// TwinCAT 3 PLC project WPPruefstand
// ProgramVersion: 3.1.4022.1
// CompilerDefines: VISU_USEPROPERTYINFO
// libraries:
//   VisuElem3DPath, 3.5.6.0 (System)
//   VisuElemMeter, 3.5.6.0 (System)
//   VisuElems, 3.5.6.10 (System)
//   VisuElemsDateTime, 3.5.6.0 (System)
//   VisuElemsSpecialControls, 3.5.6.0 (System)
//   VisuElemsWinControls, 3.5.6.0 (System)
//   VisuElemTextEditor, 3.5.6.0 (System)
//   visuinputs, 3.5.6.0 (system)
//   VisuNativeControl, 3.5.6.0 (System)
//   Tc2_Standard, * (Beckhoff Automation GmbH)
//   Tc2_System, * (Beckhoff Automation GmbH)
//   Tc2_Utilities, * (Beckhoff Automation GmbH)
//   Tc3_Module, * (Beckhoff Automation GmbH)
//   VisuDialogs, * (System)
// project tree:
//   DUTs/ E_PowMeas.TcDUT (not stored), E_Press.TcDUT (not stored), E_TempSensVR10.TcDUT (not stored), E_TempSensPT100.TcDUT (not stored), E_IndexPowMeas.TcDUT (not stored), E_SMStatus.TcDUT, E_TempSensVR11.TcDUT, E_Terminals.TcDUT (not stored), ST_InputVar.TcDUT (not stored), ST_InputVar_PowMeas.TcDUT (not stored), ST_OutputVar.TcDUT, ST_PumpTime.TcDUT
//   / GlobalTextList.TcGTLO (not stored), PlcTask.TcTTO, Visualization Manager.TcVMO (not stored)
//   GVLs/ DigOutputs.TcGVL, HeatingCurve.TcGVL, AnaOutputs.TcGVL (not stored), PID.TcGVL, PowMeas.TcGVL (not stored), Pressures.TcGVL (not stored), PumpTiming.TcGVL, StateMachine.TcGVL (not stored), SysCheck.TcGVL, SysCheckParams.TcGVL, TempConvDat.TcGVL, Temperatures.TcGVL, TempSetpoints.TcGVL, TerminalErrorRT.TcGVL, TimeProgs.TcGVL
//   POUs/ CheckDivDInt.TcPOU, CheckDivLInt.TcPOU (not stored), CheckDivLReal.TcPOU (not stored), CheckDivReal.TcPOU, MAIN.TcPOU (not stored), P_GetTime.TcPOU (not stored)
//   POUs/Control/ FB_AuxHeatCont.TcPOU (not stored), FB_CyclingControl.TcPOU, P_ControlMain.TcPOU (not stored)
//   POUs/Control/TemperatureControl/ FB_PIDSuppTemp.TcPOU, FB_SimpleTempCont.TcPOU, F_GetTempSP.TcPOU (not stored), I_TempController.TcIO (not stored), P_SHSuppTempPID.TcPOU
//   POUs/ErrorHandling/ F_WriteErrLog.TcPOU (not stored), P_EmShutdownAll.TcPOU (not stored), P_EmShutdownBPumpRun.TcPOU, P_EmShutdownHCPumpRun.TcPOU (not stored), P_EmShutdownPumpsRun.TcPOU (not stored), P_EmShutdownMain.TcPOU (not stored), P_ErrorHandlingMain.TcPOU (not stored), P_WriteErrLog.TcPOU (not stored)
//   POUs/Initialize/ FB_InitPumpTimes.TcPOU, FB_ReadHeatCurve.TcPOU, FB_ReadNightMode.TcPOU, FB_ReadPressTab.TcPOU, FB_ReadPT100Tab.TcPOU, FB_ReadTempResTabVR11.TcPOU, P_InitMain.TcPOU, FB_ReadTempResTabVR10.TcPOU, FB_InitTimes.TcPOU (not stored)
//   POUs/Read/ F_LinSens.TcPOU, F_NTCSens.TcPOU (not stored), F_PowMeasPhase.TcPOU (not stored), P_PowMeas.TcPOU, P_ReadMain.TcPOU, P_TestVals.TcPOU (not stored)
//   POUs/SystemCheck/ F_CheckAmbTemp.TcPOU (not stored), F_CheckBrinePressure.TcPOU (not stored), F_CheckCompCycPress.TcPOU, F_CheckCompOutTemp.TcPOU, F_CheckHeatCirPress.TcPOU, F_CheckHeatCirTemp.TcPOU (not stored), F_CheckPhaseSeq.TcPOU (not stored), F_CheckSens.TcPOU (not stored), F_CheckTerm.TcPOU (not stored), P_SysCheckMain.TcPOU
//   POUs/Write/ F_ConvLinAnaOutp.TcPOU (not stored), F_PumpConvPercVolt.TcPOU (not stored), FB_RampPump.TcPOU (not stored), P_WriteMain.TcPOU
//   VISUs/ Vis_ManCont.TcVIS (not stored), StandardVis.TcVIS (not stored)

CONFIGURATION WPPruefstand
    RESOURCE PLC ON TwinCAT3
        TASK PlcTask(INTERVAL := T#10ms, PRIORITY := 20);
        PROGRAM MAIN WITH PlcTask : MAIN;
    END_RESOURCE
END_CONFIGURATION

// ---- DUTs/E_SMStatus.TcDUT
{attribute 'strict'}
TYPE E_SMStatus :
(Initialize,
Read,
SystemCheck,
Automatic,
Write,
Error);
END_TYPE

// ---- DUTs/E_TempSensVR11.TcDUT
TYPE E_TempSensVR11 : //all VR11 temperature sensors
(
	T1,		//Temperature after compression
	T2,		//Temperature before compression
	T3,		//Source temperature before evaporator
	T4,		//Temperature before expansion valve
	T5,		//Temperature before internal heating circuit pump
	T6,		//Temperature after auxiliary heater
	T8		//Source temperature after brine pump
);
END_TYPE

// ---- DUTs/ST_OutputVar.TcDUT
TYPE ST_OutputVar :
STRUCT

(*
nVarOutput = (fVar-fParaC)/fParaM)
*)	

	nVarOutput AT %Q*	:INT;	//Output to terminal
	fVal				:REAL;	//Output value as REAL/FLOAT/SINGLE
	
	fParaMaxOutp		:REAL	:= 10;			//slope of linear conversion -> 10V, 32767 bit (INT16)
	nParaMaxInt			:INT	:= 32767;	
	fParaC				:REAL	:= 0;			//offset of linear conversion
	
	fParaMaxVal			:REAL;	//Maximum value of output (e.g. 10V, 20mA)
	fParaMinVal			:REAL;	//Minimum value of output (e.g. 0V, 4mA)
	
END_STRUCT
END_TYPE

// ---- DUTs/ST_PumpTime.TcDUT
TYPE ST_PumpTime :
STRUCT
	tPre	:	TIME;	//time the pump runs before compressor start
	tPost	:	TIME;	//time the pump runs after compressor stop
	bFirst	:	BOOL;	//flag if pump is the first one to start
	tDelay	:	Time;	//time the pump starts after the first pump
END_STRUCT
END_TYPE

// ---- GVLs/DigOutputs.TcGVL
{attribute 'qualified_only'}
VAR_GLOBAL
	//contactors
	bOutpComp	AT	%Q*	:	BOOL:=FALSE;	//Activate compressor - default: false
	bOutpAH		AT	%Q*	:	BOOL:=FALSE;	//Activate auxiliary heater - default: false
	
	//Switching valve
	bSHDHWSwitchValv	AT	%Q*	:	BOOL;	//Control signal for switching valve - Space Heating/DHW
	
END_VAR

// ---- GVLs/HeatingCurve.TcGVL
VAR_GLOBAL
	HeatCurve	:	ARRAY[0..40,0..1] OF REAL;
END_VAR

// ---- GVLs/PID.TcGVL
VAR_GLOBAL
	fKp			:	REAL	:= 1;		//proportional gain
	fTi			:	REAL	:= 10;		//integration time
	fTd			:	REAL	:= 0;		//derivative time
	tSamp		:	TIME	:= T#100MS;	//sampling time
	
	fErrSum		:	REAL	:= 0;	//sum of errors
	
	//limits of control signal - 0..10V signal
	fOutpUpLim	:	REAL	:=	10;
	fOutpLowLim	:	REAL	:=	0;
END_VAR

// ---- GVLs/PumpTiming.TcGVL
VAR_GLOBAL
	stBPTime			:	ST_PumpTime;
	stIntHeatCirTime	:	ST_PumpTime;
	nMaxPre				:	DWORD;
END_VAR

// ---- GVLs/SysCheck.TcGVL
VAR_GLOBAL
	bTermErrRT	:	BOOL	:=	FALSE;
	bSensErr	:	BOOL	:=	FALSE;
	bAmbTemp	:	BOOL	:=	FALSE;
	bBP			:	BOOL	:=	FALSE;
	bHCP		:	BOOL	:=	FALSE;
	bCompCyc	:	BOOL	:=	FALSE;
	bPhaseSeqCh	:	BOOL	:=	FALSE;
	bHeatTemp	:	BOOL	:=	FALSE;
	bCompOut	:	BOOL	:=	FALSE;
END_VAR

// ---- GVLs/SysCheckParams.TcGVL
VAR_GLOBAL
	(*
		All values except maximum compressor outlet temperature, maximum water supply temperature and 
		maximum water return temperature are set as recommended by the manufacturer. 
	*)	

	fMaxAmbTemp			:	REAL	:=	35;		//maximum ambient temperature
	fMinAmbTemp			:	REAL	:=	-20;	//minimum ambient temperature
	
	fBPMinOff			:	REAL	:=	0.2;	//minimum brine circuit pressure
	fBPMinOn			:	REAL	:=	0.4;	//brine circuit pressure for heat pump restart
	
	fHPMax				:	REAL	:=	30;		//maximum high pressure for compression cycle
	fLPMin				:	REAL	:=	0.7;	//minimum low pressure for compression cycle
	
	fTempCompOutMax		:	REAL	:=	120;	//maximum compressor outlet temperature
	
	fHCPMinOff			:	REAL	:=	0.5;	//minimum heating circuit pressure
	fHCPMinOn			:	REAL	:=	0.7;	//heating circuit pressure for heat pump restart
	
	fTempHeatSuppMax	:	REAL	:=	65;		//maximum water supply temperature
	fTempHeatRetMax		:	REAL	:=	60;		//maximum water return temperature
END_VAR

// ---- GVLs/TempConvDat.TcGVL
VAR_GLOBAL
	//stTempSensTables	:	ST_TempSensTables;
	VR10	:	ARRAY[1..40,1..2] OF REAL;
	VR11	:	ARRAY[1..40,1..2] OF REAL;
END_VAR

// ---- GVLs/Temperatures.TcGVL
{attribute 'qualified_only'}
VAR_GLOBAL
	eTempSensVR10	:	E_TempSensVR10;	//VR10 temperature sensors
	eTempSensVR11	:	E_TempSensVR11;	//VR11 temperature sensors
	eTempSensPT100	:	E_TempSensPT100;	//PT100 temperature sensors
	
	stTempSensVR10	:	ARRAY[0..3] OF ST_InputVar;	//Structures corresponding to temperature sensor enumeration
	stTempSensVR11	:	ARRAY[0..6] OF ST_InputVar;
	stTempSensPT100	:	ARRAY[0..3] OF ST_InputVar;

(*
	//Internal temperature sensors
	//Names of temperatures according to installation manual
	stT1	:	ST_InputVar;	//Temperature after compression
	stT2	:	ST_InputVar;	//Temperature before compression
	stT3	:	ST_InputVar;	//Source temperature before evaporator
	stT4	:	ST_InputVar;	//Temperature before expansion valve
	stT5	:	ST_InputVar;	//Temperature before internal heating circuit pump
	stT6	:	ST_InputVar;	//Temperature after auxiliary heater
	stT8	:	ST_InputVar;	//Source temperature after brine pump
	stSP	:	ST_InputVar;	//Temperature of DHW storage tank
	stVF1	:	ST_InputVar;	//Temperature at the top of the space heating buffer tank
	stVF2	:	ST_InputVar;	//Temperature after external mixing valve
	stRF1	:	ST_InputVar;	//Temperature at the bottom of the space heating buffer tank
	
	//Additional temperature sensors
	stTEXPVEV	:	ST_InputVar;	//Temperature between expansion valve and evaporator
	stTSHEV		:	ST_InputVar;	//Temperature after evaporator
	stTCond		:	ST_InputVar;	//Temperature after condenser
	stTAmp		:	ST_InputCar;	//Ambient temperature
*)

END_VAR

// ---- GVLs/TempSetpoints.TcGVL
VAR_GLOBAL
	fDHWUpSP			:	REAL	:=	65;	//hot water temperature upper setpoint for DHW
	fDHWLowSP			:	REAL	:=	55;	//hot water temperature lower setpoint for DHW
	fSpaceHeatSP		:	REAL;			//water supply temperature setpoint for space heating
	fRoomSetpoint		:	REAL	:=	20;	//room temperature setpoint temperature
	fRoomSetpointNight	:	REAL	:=	15;	//room temperature setpoint for night mode
END_VAR

// ---- GVLs/TerminalErrorRT.TcGVL
VAR_GLOBAL
	//check if the real-time communication with the terminals reports errors
	//checks State of Working Counter: 
	//0 - valid real-time communication
	//1 - invalid real-time communication
	bTermRt		AT %I*	:	ARRAY[0..8] OF BOOL;
END_VAR

// ---- GVLs/TimeProgs.TcGVL
VAR_GLOBAL
	todNightModeStart	:	TOD;
	todNightModeEnd		:	TOD;
END_VAR

// ---- POUs/CheckDivDInt.TcPOU
// Implicitly generated code : DO NOT EDIT
FUNCTION CheckDivDInt : DINT
VAR_INPUT
	divisor:DINT;
END_VAR

// Implicitly generated code : Only an Implementation suggestion
IF divisor = 0 THEN
	CheckDivDInt:=1;
	StateMachine.bFault		:=	TRUE;
	StateMachine.nFault		:=	2;
	StateMachine.sFaultMess	:=	'Critical program error: division by 0';
	StateMachine.eStatus	:=	Error;
	P_EmShutdownAll();	//Execute emergency shutdown
ELSE
	CheckDivDInt:=divisor;
END_IF;

END_FUNCTION

// ---- POUs/CheckDivReal.TcPOU
// Implicitly generated code : DO NOT EDIT
FUNCTION CheckDivReal : REAL
VAR_INPUT
	divisor:REAL;
END_VAR

// Implicitly generated code : Only an Implementation suggestion
IF divisor = 0 THEN
	CheckDivReal:=1;
	StateMachine.bFault		:=	TRUE;
	StateMachine.nFault		:=	2;
	StateMachine.sFaultMess	:=	'Critical program error: division by 0';
	StateMachine.eStatus	:=	Error;
	P_EmShutdownAll();	//Execute emergency shutdown
ELSE
	CheckDivReal:=divisor;
END_IF;

END_FUNCTION

// ---- POUs/Control/FB_CyclingControl.TcPOU
FUNCTION_BLOCK FB_CyclingControl
VAR_INPUT
	nMaxStarts	:	USINT	:=	3;		//maximum number of startups per hour
	nMinRunTime	:	DWORD	:=	300;	//minimum run time in seconds
	nMinOffTime	:	DWORD	:=	300;	//minimum off time in seconds
END_VAR
VAR_OUTPUT
	bStartupOK	:	BOOL;
	bShutdownOK	:	BOOL;
END_VAR
VAR
	//Startup counter
	TimHour		:	TON;	//timer for 1h
	
	//run time | off time
	nLastStart	:	DWORD;
	nLastStop	:	DWORD;
	
	//Current time
	nCurTime	:	DWORD;
	
END_VAR

//Timer parameters
TimHour.PT	:=	T#1h;
TimHour.IN	:=	TRUE;
TimHour();
IF TimHour.Q THEN			//one hour has passed
	TimHour.IN	:=	FALSE;	//reset timer
	TimHour();
	StateMachine.nNumStart	:=	0;		//reset counter
END_IF

//last start and stop time in seconds
nLastStart	:=	DT_TO_DWORD(StateMachine.dtLastStart);
nLastStop	:=	DT_TO_DWORD(StateMachine.dtLastStop);

//Current time
nCurTime	:=	DT_TO_DWORD(StateMachine.dtCurTime);	//current time in seconds

//set startup flag
IF (StateMachine.nNumStart >= nMaxStarts) OR (NOT ((nCurTime - nLastStop) >= (nMinOffTime - PumpTiming.nMaxPre))) THEN
	//disable startup, if max. starts per hour are reached or minimum off time is violated
	bSTartupOK	:=	FALSE;
ELSE
	bStartupOK	:=	TRUE;
END_IF

//set shutdown flag
IF NOT ((nCurTime - nLastStart) >= nMinRunTime) THEN
	bShutdownOK :=	FALSE;
ELSE
	bShutdownOK :=	TRUE;
END_IF

END_FUNCTION_BLOCK

// ---- POUs/Control/TemperatureControl/FB_PIDSuppTemp.TcPOU
FUNCTION_BLOCK FB_PIDSuppTemp
VAR_INPUT
	fSetPoint	:	REAL;
END_VAR
VAR_OUTPUT
	fOutp		:	REAL;
END_VAR
VAR
	Tim			:	TON;
	
	fErr		:	REAL;			//current difference between setpoint and actual value
	fErrOld		:	REAL	:= 0;	//error in last cycle
	
	eVF2		:	E_TempSensVR10	:=	VF2;
END_VAR

Tim(PT:=PID.tSamp,IN:=TRUE);

IF Tim.Q THEN
	//calculate current difference
	fErr	:=	fSetPoint - Temperatures.stTempSensVR10[eVF2].fVal;

	//Anti-windup
	IF (fOutp < PID.fOutpUpLim) AND (fOutp > PID.fOutpLowLim) THEN
		PID.fErrSum	:=	PID.fErrSum + (fErr * (TIME_TO_REAL(PID.tSamp)/1000));	//Integrate
	END_IF

	//calculate output signal
	fOutp	:=	PID.fKp * (fErr + (1/PID.fTi) * PID.fErrSum + PID.fTd * ((fErr - fErrOld)/(TIME_TO_REAL(PID.tSamp) / 1000)));

	IF fOutp > PID.fOutpUpLim THEN
		fOutp	:= PID.fOutpUpLim;
	ELSIF fOutp < PID.fOutpLowLim THEN
		fOutp	:=	PID.fOutpLowLim;
	END_IF

	//save error
	fErrOld	:=	fErr;
	
	//reset timer
	Tim(IN:=FALSE);
END_IF

END_FUNCTION_BLOCK

// ---- POUs/Control/TemperatureControl/FB_SimpleTempCont.TcPOU
FUNCTION_BLOCK FB_SimpleTempCont IMPLEMENTS I_TempController
VAR_INPUT
	//maximum times
	tMaxTimeDHW		:	TIME	:=	T#40M;
	tMaxTimeSH		:	TIME	:=	T#20M;
END_VAR
VAR_OUTPUT
END_VAR
VAR
	eSP				:	E_TempSensVR10	:=	SP;
	eRF1			:	E_TempSensVR10	:=	RF1;
	eVF1			:	E_TempSensVR10	:=	VF1;
	eAmb			:	E_TempSensPT100	:=	TAmb;
	
	//flags demand
	bDemDHW			:	BOOL	:=	FALSE;	//DHW demand
	bDemSH			:	BOOL	:=	FALSE;	//Space heating demand
	bEarlyRech		:	BOOL	:=	FALSE;	//early recharching of space heating buffer tank
	
	//timers for parallel demand
	TimDHW			:	TON;
	TimSH			:	TON;
	
	//Compressor control values
	CompOpCont		:	BOOL	:=	FALSE;
	ValveModeCont	:	BOOL;
	
	fSHTempSP		:	REAL;
END_VAR

//get temperature setpoint from heating curve
fSHTempSP	:=	F_GetTempSP(fAmbTemp:=Temperatures.stTempSensPT100[eAmb].fVal);

//identify DHW demand
IF (Temperatures.stTempSensVR10[eSP].fVal < TempSetpoints.fDHWLowSP) THEN
	bDemDHW		:=	TRUE;	//temperature lower than low setpoint -> demand
END_IF
IF (Temperatures.stTempSensVR10[eSP].fVal > TempSetpoints.fDHWUpSP) THEN
	IF ((Temperatures.stTempSensVR10[eVF1].fVal < (TempSetpoints.fSpaceHeatSP + 2))) AND bDemDHW THEN
		bEarlyRech	:=	TRUE;
	END_IF
	bDemDHW	:=	FALSE;	//temperature higher than upper setpoint -> cancel demand
END_IF

//identify space heating demand
IF (Temperatures.stTempSensVR10[eVF1].fVal < TempSetpoints.fSpaceHeatSP) THEN
	bDemSH		:=	TRUE;
END_IF
IF (Temperatures.stTempSensVR10[eRF1].fVal > (TempSetpoints.fSpaceHeatSP + 2)) THEN
	bDemSH		:=	FALSE;
END_IF
IF (Temperatures.stTempSensVR10[eRF1].fVal > (TempSetpoints.fSpaceHeatSP + 2)) THEN
	bEarlyRech	:=	FALSE;
END_IF

//Set modes

//Switching valve mode: 
//True: space heating mode
//False: DHW mode	
IF bDemDHW AND (NOT bDemSH) THEN			//only DHW demand
	ValveModeCont	:=	FALSE;
	CompOpCont		:=	TRUE;
ELSIF bDemSH AND (NOT bDemDHW) THEN			//only space heating demand
	ValveModeCont	:=	TRUE;
	CompOpCont		:=	TRUE;
ELSIF (NOT bDemSH) AND (NOT bDemDHW) THEN	//no demand
	IF bEarlyRech THEN	//early recharging
		ValveModeCont	:=	TRUE;
		CompOpCont		:=	TRUE;
	ELSE
		CompOpCont		:=	FALSE;
	END_IF
ELSIF bDemSH AND bDemDHW THEN				//parallel demand
	CompOpCont		:= TRUE;
	IF (NOT ValveModeCont) AND TimDHW.Q THEN	//max. time DHW mode reached
		ValveModeCont	:=	TRUE;	//switch to space heating
	ELSIF ValveModeCont AND TimSH.Q THEN		//max. time SH mode reached
		ValveModeCont	:=	FALSE;	//switch to DHW
	END_IF	
END_IF

//Timing
TimDHW.PT	:=	tMaxTimeDHW;
TImSH.PT	:=	tMaxTimeSH;
TimDHW();
TimSH();
IF StateMachine.bCompRun THEN	//only when the compressor is actually running
	IF ValveModeCont THEN
		TimSH.IN	:=	TRUE;
		TimDHW.IN	:=	FALSE;
	ELSE
		TimSH.IN	:=	FALSE;
		TimDHW.IN	:=	TRUE;
	END_IF
ELSE
	TimSH.IN		:=	FALSE;
	TimDHW.IN		:=	FALSE;
END_IF

PROPERTY CompOp : BOOL
GET
CompOp	:=	CompOpCont;
END_GET
SET
CompOpCont	:=	CompOp;
END_SET
END_PROPERTY

PROPERTY SpaceHeatTempSP : REAL
GET
SpaceHeatTempSP	:=	fSHTempSP;
END_GET
SET
fSHTempSP	:=	SpaceHeatTempSP;
END_SET
END_PROPERTY

PROPERTY ValveMode : BOOL
GET
ValveMode	:=	ValveModeCont;
END_GET
SET
ValveModeCont	:= ValveMode;
END_SET
END_PROPERTY

END_FUNCTION_BLOCK

// ---- POUs/Control/TemperatureControl/P_SHSuppTempPID.TcPOU
PROGRAM P_SHSuppTempPID
VAR
	eTAmb			:	E_TempSensPT100	:=	TAmb;	//ambient temperature
	fTAmbMax		:	REAL			:=	21;		//maximum ambient temperature before space heating is switched off
	fbPIDSuppTemp	:	FB_PIDSuppTemp;				//PID controller
	fPIDOutp		:	REAL;						//control signal from PID
	bAct			:	BOOL			:=	True;	//space heating active
END_VAR

IF Temperatures.stTempSensPT100[eTAmb].fVal > (fTAmbMax + 1) THEN
	bAct	:=	FALSE;
ELSIF Temperatures.stTempSensPT100[eTAmb].fVal < (fTAmbMax - 1) THEN
	bAct	:=	TRUE;
END_IF
	
IF bAct THEN
	//run external heating circuit pump
	StateMachine.bExtHeatCPump	:=	TRUE;

	//execute PID Control
	fbPIDSuppTemp(fSetPoint:=TempSetpoints.fSpaceHeatSP);
	fPIDOutp	:=	fbPIDSuppTemp.fOutp;

	//pass control signal to mixing valve
	StateMachine.fMixVal	:=	fPIDOutp;
ELSE
	StateMachine.bExtHeatCPump	:=	FALSE;
END_IF

END_PROGRAM

// ---- POUs/ErrorHandling/P_EmShutdownBPumpRun.TcPOU
PROGRAM P_EmShutdownBPumpRun
VAR
END_VAR

//shut down all components except brine pump

StateMachine.bCompRun		:=	FALSE;
DigOutputs.bOutpComp		:=	FALSE;

StateMachine.bAuxHeatOp		:=	FALSE;
DigOutputs.bOutpAH			:=	FALSE;

StateMachine.bBrinePump		:=	TRUE;
AnaOutputs.stOutpBP.fVal	:=	10;
AnaOutputs.stOutpBP			:=	F_ConvLinAnaOutp(stOutput:=AnaOutputs.stOutpBP);

StateMachine.bIntHeatCPump	:=	FALSE;
AnaOutputs.stOutpIntHP.fVal	:=	0.75;	//0.75 Volt: Pump stop
AnaOutputs.stOutpIntHP		:=	F_ConvLinAnaOutp(stOutput:=AnaOutputs.stOutpIntHP);

StateMachine.bExtHeatCPump	:=	TRUE;
AnaOutputs.stOutpExtHP.fVal	:=	10;	
AnaOutputs.stOutpExtHP			:=	F_ConvLinAnaOutp(stOutput:=AnaOutputs.stOutpExtHP);

StateMachine.bCircPump		:=	TRUE;

END_PROGRAM

// ---- POUs/Initialize/FB_InitPumpTimes.TcPOU
FUNCTION_BLOCK FB_InitPumpTimes
VAR_INPUT
	tBP_Pre				:	TIME	:=	T#1M;
	tIntHeatCir_Pre		:	TIME	:=	T#1M;
	tBP_Post			:	TIME	:=	T#5M;
	tIntHeatCir_Post	:	TIME	:=	T#30M;
END_VAR
VAR_OUTPUT
	bReady	:	BOOL	:=	False;
END_VAR
VAR
END_VAR

//write to GVL
PumpTiming.stBPTime.tPre			:=	tBP_Pre;
PumpTiming.stIntHeatCirTime.tPre	:=	tIntHeatCir_Pre;
PumpTiming.stBPTime.tPost			:=	tBP_Post;
PumpTiming.stIntHeatCirTime.tPost	:=	tIntHeatCir_Post;

//find first one to start and calculate delays
IF (tBP_Pre > tIntHeatCir_Pre) THEN
	PumpTiming.stBPTime.bFirst			:=	TRUE;
	PumpTiming.stBPTime.tDelay			:=	T#0MS;
	PumpTiming.stIntHeatCirTime.tDelay	:=	tBP_Pre - tIntHeatCir_Pre;
	PumpTiming.nMaxPre					:=	(TIME_TO_DWORD(tBP_Pre)/1000);
ELSE
	PumpTiming.stIntHeatCirTime.bFirst	:=	TRUE;
	PumpTiming.stIntHeatCirTime.tDelay	:=	T#0MS;
	PumpTiming.stBPTime.tDelay			:=	tIntHeatCir_Pre - tBP_Pre;
	PumpTiming.nMaxPre					:=	(TIME_TO_DWORD(tIntHeatCir_Pre)/1000);
END_IF

bReady	:=	TRUE;

END_FUNCTION_BLOCK

// ---- POUs/Initialize/FB_ReadHeatCurve.TcPOU
FUNCTION_BLOCK FB_ReadHeatCurve
VAR_INPUT
	bExecute		:	BOOL	:= FALSE;
END_VAR
VAR_OUTPUT
	bCompleted		:	BOOL	:=	FALSE;
	bError			:	BOOL	:=	FALSE;
END_VAR
VAR
	fbFileOpen		:	FB_FileOpen;
	fbFileGets		:	FB_FileGets;
	fbReader		:	FB_CSVMemBufferReader;
	fbFileClose		:	FB_FileClose;
	sCSVPath		:	STRING	:=	'D:\cve-mme\WpPruefstandData\Heizkurve.csv';	//Path to csv file
	hFile			:	UINT;
	bEOF			:	BOOL	:=	FALSE;
	Step			:	DWORD	:=	0;
	sLine			:	STRING;	//Line read by fbFileGets
	nLine			:	UINT	:=	0;
END_VAR

CASE Step OF
	
0:	//Standby mode
	IF bExecute THEN
		bExecute	:=	FALSE; //reset to defaults
		hFile		:=	0;
		bEOF		:=	FALSE;
		bCompleted	:=	FALSE;
		bError		:=	FALSE;
		sLine		:=	'';
		nLine		:=	0;
		Step		:=	1; //start program
	END_IF

1:	//Open file
	fbFileOpen(sNetId:='', sPathName:=sCSVPath, nMode:=FOPEN_MODEREAD OR FOPEN_MODETEXT,
		ePath:=PATH_GENERIC, tTimeout:=T#5s, bExecute:=TRUE);
	Step	:=	Step + 1;

2:
	fbFileOpen(bExecute:=FALSE);
	IF NOT fbFileOpen.bBusy THEN
		IF NOT fbFileOpen.bError THEN
			//Store file handle
			hFile	:=	fbFileOpen.hFile;
			Step	:=	Step + 1;
		ELSE
			Step	:=	90;	
		END_IF
	END_IF

3:	//Read csv file
	fbFileGets(sNetId:='', hFile:=hFile, bExecute:=TRUE, tTimeout:=T#5S);
	nLine	:=	nLine + 1;
	Step	:=	Step + 1;

4:
	fbFileGets(bExecute:=FALSE);
	IF NOT fbFileGets.bBusy THEN
		IF NOT (nLine = 1) THEN //Header -> jump to next line
			IF NOT fbFileGets.bError THEN
				IF fbFileGets.bEOF THEN
					Step	:=	10; //Reached end of file
				ELSE
					sLine	:=	fbFileGets.sLine; //store line
					IF RIGHT(sLine,1) = '$L' THEN
						sLine	:=	REPLACE(sLINE, '$R$L', 2, LEN(sLine)); //restore CRLF characters
					END_IF
					Step	:=	Step + 1;
				END_IF
			ELSE
				Step	:=	90;
			END_IF
		ELSE
			Step	:=	3;
		END_IF
	END_IF
	
5:	//Parse line
	
	fbReader.eCmd	:=	eEnumCmd_First;	//Read first value (ambient temperature)
	fbReader(pBuffer:=ADR(sLine), cbBuffer:=SIZEOF(sLine));
	
	IF fbReader.bOk THEN
		HeatingCurve.HeatCurve[nLine-2,0] := STRING_TO_REAL(fbReader.getValue);	//account for header
	ELSE
		Step	:=	90;
	END_IF	
	
	fbReader.eCmd	:=	eEnumCmd_Next;	//Read next value (temperature setpoint)
	fbReader(pBuffer:=ADR(sLine), cbBuffer:=SIZEOF(sLine));
	
	IF fbReader.bOk THEN
		HeatingCurve.HeatCurve[nLine-2,1] := STRING_TO_REAL(fbReader.getValue); //account for header
	ELSE
		Step	:=	90;
	END_IF
	
	//Read next line
	Step	:=	3;
	
10:	//end of csv file
	IF (hFile <> 0) THEN
		Step	:=	20; //close file
	END_IF
	
20:	//close csv file
	fbFileClose(bExecute:=FALSE);
	fbFileClose(sNetId:='', hFile:=hFile, bExecute:=TRUE, tTimeout:=T#5S);
	Step	:=	21;
	
21:	
	fbFileClose(bExecute:=FALSE);
	IF NOT fbFileClose.bBusy THEN
		step	:=	0;	//Standby mode
		bCompleted	:=	TRUE;
	END_IF
	
90:	//TODO: Error handling
	bError	:=	TRUE;
	IF (hFile <> 0) THEN
		Step	:=	20;	//close file
	END_IF

END_CASE

END_FUNCTION_BLOCK

// ---- POUs/Initialize/FB_ReadNightMode.TcPOU
FUNCTION_BLOCK FB_ReadNightMode
VAR_INPUT
	bExecute		:	BOOL	:= FALSE;
END_VAR
VAR_OUTPUT
	bCompleted		:	BOOL	:=	FALSE;
	bError			:	BOOL	:=	FALSE;
END_VAR
VAR
	fbFileOpen		:	FB_FileOpen;
	fbFileGets		:	FB_FileGets;
	fbReader		:	FB_CSVMemBufferReader;
	fbFileClose		:	FB_FileClose;
	sCSVPath		:	STRING	:=	'D:\cve-mme\WpPruefstandData\NightMode.csv';	//Path to csv file
	hFile			:	UINT;
	bEOF			:	BOOL	:=	FALSE;
	Step			:	DWORD	:=	0;
	sLine			:	STRING;	//Line read by fbFileGets
	nLine			:	UINT	:=	0;
	nHourStart		:	USINT;
	nHourStop		:	USINT;
	nMinStart		:	USINT;
	nMinStop		:	USINT;
	nStartTime		:	UDINT;	//Start time in ms
	nStopTime		:	UDINT;	//Stop time in ms
END_VAR

CASE Step OF
	
0:	//Standby mode
	IF bExecute THEN
		bExecute	:=	FALSE; //reset to defaults
		hFile		:=	0;
		bEOF		:=	FALSE;
		bCompleted	:=	FALSE;
		bError		:=	FALSE;
		sLine		:=	'';
		nLine		:=	0;
		Step		:=	1; //start program
	END_IF

1:	//Open file
	fbFileOpen(sNetId:='', sPathName:=sCSVPath, nMode:=FOPEN_MODEREAD OR FOPEN_MODETEXT,
		ePath:=PATH_GENERIC, tTimeout:=T#5s, bExecute:=TRUE);
	Step	:=	Step + 1;

2:
	fbFileOpen(bExecute:=FALSE);
	IF NOT fbFileOpen.bBusy THEN
		IF NOT fbFileOpen.bError THEN
			//Store file handle
			hFile	:=	fbFileOpen.hFile;
			Step	:=	Step + 1;
		ELSE
			Step	:=	90;	
		END_IF
	END_IF

3:	//Read csv file
	fbFileGets(sNetId:='', hFile:=hFile, bExecute:=TRUE, tTimeout:=T#5S);
	nLine	:=	nLine + 1;
	Step	:=	Step + 1;

4:
	fbFileGets(bExecute:=FALSE);
	IF NOT fbFileGets.bBusy THEN
		IF NOT (nLine = 1) THEN //Header -> jump to next line
			IF NOT fbFileGets.bError THEN
				IF fbFileGets.bEOF THEN
					Step	:=	10; //Reached end of file
				ELSE
					sLine	:=	fbFileGets.sLine; //store line
					IF RIGHT(sLine,1) = '$L' THEN
						sLine	:=	REPLACE(sLINE, '$R$L', 2, LEN(sLine)); //restore CRLF characters
					END_IF
					Step	:=	Step + 1;
				END_IF
			ELSE
				Step	:=	90;
			END_IF
		ELSE
			Step	:=	3;
		END_IF
	END_IF
	
5:	//Parse line
	fbReader.eCmd	:=	eEnumCmd_First;	//Read first value (identifier)
	fbReader(pBuffer:=ADR(sLine), cbBuffer:=SIZEOF(sLine));
	
	fbReader.eCmd	:=	eEnumCmd_Next;	//Read next value (hour)
	fbReader(pBuffer:=ADR(sLine), cbBuffer:=SIZEOF(sLine));
	
	IF fbReader.bOk THEN
		IF (nLine = 2) THEN
			nHourStart	:=	STRING_TO_USINT(fbReader.getValue);
		ELSIF (nLine = 3) THEN
			nHourStop	:=	STRING_TO_USINT(fbReader.getValue);
		ELSE
			Step	:=	90;
		END_IF
	ELSE
		Step	:=	90;
	END_IF	
	
	fbReader.eCmd	:=	eEnumCmd_Next;	//Read next value (minute)
	fbReader(pBuffer:=ADR(sLine), cbBuffer:=SIZEOF(sLine));
	
	IF fbReader.bOk THEN
		IF (nLine = 2) THEN
			nMinStart	:=	STRING_TO_USINT(fbReader.getValue);
		ELSIF (nLine = 3) THEN
			nMinStop	:=	STRING_TO_USINT(fbReader.getValue);
		ELSE
			Step	:=	90;
		END_IF
	ELSE
		Step	:=	90;
	END_IF
	
	//Read next line
	Step	:=	3;
	
10:	//end of csv file
	IF (hFile <> 0) THEN
		Step	:=	20; //close file
	END_IF
	
20:	//close csv file
	fbFileClose(bExecute:=FALSE);
	fbFileClose(sNetId:='', hFile:=hFile, bExecute:=TRUE, tTimeout:=T#5S);
	Step	:=	21;
	
21:	
	fbFileClose(bExecute:=FALSE);
	IF NOT fbFileClose.bBusy THEN
		//convert data and write to GVL
		nStartTime	:=	nHourStart * 3600 * 1000 + nMinStart * 60 * 1000;
		nStopTime	:=	nHourStop * 3600 * 1000 + nMinStop * 60 * 1000;
		TimeProgs.todNightModeStart	:=	UDINT_TO_TOD(nStartTime);
		TimeProgs.todNightModeEnd	:=	UDINT_TO_TOD(nStopTime);
	
		step	:=	0;	//Standby mode
		bCompleted	:=	TRUE;
	END_IF
	
90:	//TODO: Error handling
	bError	:=	TRUE;
	IF (hFile <> 0) THEN
		Step	:=	20;	//close file
	END_IF

END_CASE

END_FUNCTION_BLOCK

// ---- POUs/Initialize/FB_ReadPressTab.TcPOU
FUNCTION_BLOCK FB_ReadPressTab
VAR_INPUT
	bExecute		:	BOOL	:= FALSE;
END_VAR
VAR_OUTPUT
	bCompleted		:	BOOL	:=	FALSE;
	bError			:	BOOL	:=	FALSE;
END_VAR
VAR
	fbFileOpen		:	FB_FileOpen;
	fbFileGets		:	FB_FileGets;
	fbReader		:	FB_CSVMemBufferReader;
	fbFileClose		:	FB_FileClose;
	sCSVPath		:	STRING	:=	'D:\cve-mme\WpPruefstandData\PressureDat.csv';	//Path to csv file
	hFile			:	UINT;
	bEOF			:	BOOL	:=	FALSE;
	Step			:	DWORD	:=	0;
	sLine			:	STRING;	//Line read by fbFileGets
	nLine			:	UINT	:=	0;
	nIndSens		:	INT;
	stSensName		:	String;
END_VAR

CASE Step OF
	
0:	//Standby mode
	IF bExecute THEN
		bExecute	:=	FALSE; //reset to defaults
		hFile		:=	0;
		bEOF		:=	FALSE;
		bCompleted	:=	FALSE;
		bError		:=	FALSE;
		sLine		:=	'';
		nLine		:=	0;
		Step		:=	1; //start program
	END_IF

1:	//Open file
	fbFileOpen(sNetId:='', sPathName:=sCSVPath, nMode:=FOPEN_MODEREAD OR FOPEN_MODETEXT,
		ePath:=PATH_GENERIC, tTimeout:=T#5s, bExecute:=TRUE);
	Step	:=	Step + 1;

2:
	fbFileOpen(bExecute:=FALSE);
	IF NOT fbFileOpen.bBusy THEN
		IF NOT fbFileOpen.bError THEN
			//Store file handle
			hFile	:=	fbFileOpen.hFile;
			Step	:=	Step + 1;
		ELSE
			Step	:=	90;	
		END_IF
	END_IF

3:	//Read csv file
	fbFileGets(sNetId:='', hFile:=hFile, bExecute:=TRUE, tTimeout:=T#5S);
	nLine	:=	nLine + 1;
	Step	:=	Step + 1;

4:
	fbFileGets(bExecute:=FALSE);
	IF NOT fbFileGets.bBusy THEN
		IF NOT (nLine = 1) THEN //Header -> jump to next line
			IF NOT fbFileGets.bError THEN
				IF fbFileGets.bEOF THEN
					Step	:=	10; //Reached end of file
				ELSE
					sLine	:=	fbFileGets.sLine; //store line
					IF RIGHT(sLine,1) = '$L' THEN
						sLine	:=	REPLACE(sLINE, '$R$L', 2, LEN(sLine)); //restore CRLF characters
					END_IF
					Step	:=	Step + 1;
				END_IF
			ELSE
				Step	:=	90;
			END_IF
		ELSE
			Step	:=	3;
		END_IF
	END_IF
	
5:	//Parse line
	fbReader.eCmd	:=	eEnumCmd_First;	//Read first value (identifier)
	fbReader(pBuffer:=ADR(sLine), cbBuffer:=SIZEOF(sLine));
	
	IF fbReader.bOk THEN
		stSensName	:= fbReader.getValue;	//identify index of current sensor
		IF (FIND(str1:=stSensName, str2:='HP') <> 0) THEN
			Pressures.ePress	:=	HP;
		ELSIF (FIND(str1:=stSensName, str2:='LP') <> 0) THEN
			Pressures.ePress	:=	LP;
		ELSIF (FIND(str1:=stSensName, str2:='HCP') <> 0) THEN
			Pressures.ePress	:=	HCP;
		ELSIF (FIND(str1:=stSensName, str2:='BP') <> 0) THEN
			Pressures.ePress	:=	BP;
		END_IF
		nIndSens	:=	Pressures.ePress;
	ELSE
		Step	:=	90;
	END_IF	
	
	fbReader.eCmd	:=	eEnumCmd_Next;	//Read next value (slope)
	fbReader(pBuffer:=ADR(sLine), cbBuffer:=SIZEOF(sLine));
	
	IF fbReader.bOk THEN
		Pressures.stPress[nIndSens].fParaM := STRING_TO_REAL(fbReader.getValue);
	ELSE
		Step	:=	90;
	END_IF	
	
	fbReader.eCmd	:=	eEnumCmd_Next;	//Read next value (offset)
	fbReader(pBuffer:=ADR(sLine), cbBuffer:=SIZEOF(sLine));
	
	IF fbReader.bOk THEN
		Pressures.stPress[nIndSens].fParaC := STRING_TO_REAL(fbReader.getValue); //account for header
	ELSE
		Step	:=	90;
	END_IF
	
	fbReader.eCmd	:=	eEnumCmd_Next;	//Read next value (maximum value)
	fbReader(pBuffer:=ADR(sLine), cbBuffer:=SIZEOF(sLine));
	
	IF fbReader.bOk THEN
		Pressures.stPress[nIndSens].fParaMaxVal := STRING_TO_REAL(fbReader.getValue); //account for header
	ELSE
		Step	:=	90;
	END_IF
	
	fbReader.eCmd	:=	eEnumCmd_Next;	//Read next value (minimum value)
	fbReader(pBuffer:=ADR(sLine), cbBuffer:=SIZEOF(sLine));
	
	IF fbReader.bOk THEN
		Pressures.stPress[nIndSens].fParaMinVal := STRING_TO_REAL(fbReader.getValue); //account for header
	ELSE
		Step	:=	90;
	END_IF
	
	//Read next line
	Step	:=	3;
	
10:	//end of csv file
	IF (hFile <> 0) THEN
		Step	:=	20; //close file
	END_IF
	
20:	//close csv file
	fbFileClose(bExecute:=FALSE);
	fbFileClose(sNetId:='', hFile:=hFile, bExecute:=TRUE, tTimeout:=T#5S);
	Step	:=	21;
	
21:	
	fbFileClose(bExecute:=FALSE);
	IF NOT fbFileClose.bBusy THEN
		step	:=	0;	//Standby mode
		bCompleted	:=	TRUE;
	END_IF
	
90:	//TODO: Error handling
	bError	:=	TRUE;
	IF (hFile <> 0) THEN
		Step	:=	20;	//close file
	END_IF

END_CASE

END_FUNCTION_BLOCK

// ---- POUs/Initialize/FB_ReadPT100Tab.TcPOU
FUNCTION_BLOCK FB_ReadPT100Tab
VAR_INPUT
	bExecute		:	BOOL	:= FALSE;
END_VAR
VAR_OUTPUT
	bCompleted		:	BOOL	:=	FALSE;
	bError			:	BOOL	:=	FALSE;
END_VAR
VAR
	fbFileOpen		:	FB_FileOpen;
	fbFileGets		:	FB_FileGets;
	fbReader		:	FB_CSVMemBufferReader;
	fbFileClose		:	FB_FileClose;
	sCSVPath		:	STRING	:=	'D:\cve-mme\WpPruefstandData\PT100Dat.csv';	//Path to csv file
	hFile			:	UINT;
	bEOF			:	BOOL	:=	FALSE;
	Step			:	DWORD	:=	0;
	sLine			:	STRING;	//Line read by fbFileGets
	nLine			:	UINT	:=	0;
	nIndSens		:	INT;
	stSensName		:	String;
END_VAR

CASE Step OF
	
0:	//Standby mode
	IF bExecute THEN
		bExecute	:=	FALSE; //reset to defaults
		hFile		:=	0;
		bEOF		:=	FALSE;
		bCompleted	:=	FALSE;
		bError		:=	FALSE;
		sLine		:=	'';
		nLine		:=	0;
		Step		:=	1; //start program
	END_IF

1:	//Open file
	fbFileOpen(sNetId:='', sPathName:=sCSVPath, nMode:=FOPEN_MODEREAD OR FOPEN_MODETEXT,
		ePath:=PATH_GENERIC, tTimeout:=T#5s, bExecute:=TRUE);
	Step	:=	Step + 1;

2:
	fbFileOpen(bExecute:=FALSE);
	IF NOT fbFileOpen.bBusy THEN
		IF NOT fbFileOpen.bError THEN
			//Store file handle
			hFile	:=	fbFileOpen.hFile;
			Step	:=	Step + 1;
		ELSE
			Step	:=	90;	
		END_IF
	END_IF

3:	//Read csv file
	fbFileGets(sNetId:='', hFile:=hFile, bExecute:=TRUE, tTimeout:=T#5S);
	nLine	:=	nLine + 1;
	Step	:=	Step + 1;

4:
	fbFileGets(bExecute:=FALSE);
	IF NOT fbFileGets.bBusy THEN
		IF NOT (nLine = 1) THEN //Header -> jump to next line
			IF NOT fbFileGets.bError THEN
				IF fbFileGets.bEOF THEN
					Step	:=	10; //Reached end of file
				ELSE
					sLine	:=	fbFileGets.sLine; //store line
					IF RIGHT(sLine,1) = '$L' THEN
						sLine	:=	REPLACE(sLINE, '$R$L', 2, LEN(sLine)); //restore CRLF characters
					END_IF
					Step	:=	Step + 1;
				END_IF
			ELSE
				Step	:=	90;
			END_IF
		ELSE
			Step	:=	3;
		END_IF
	END_IF
	
5:	//Parse line
	fbReader.eCmd	:=	eEnumCmd_First;	//Read first value (identifier)
	fbReader(pBuffer:=ADR(sLine), cbBuffer:=SIZEOF(sLine));
	
	IF fbReader.bOk THEN
		stSensName	:= fbReader.getValue;	//identify index of current sensor
		IF (FIND(str1:=stSensName, str2:='TExpVEv') <> 0) THEN
			Temperatures.eTempSensPT100	:=	TExpVEv;
		ELSIF (FIND(str1:=stSensName, str2:='TShEv') <> 0) THEN
			Temperatures.eTempSensPT100	:=	TShEv;
		ELSIF (FIND(str1:=stSensName, str2:='TCond') <> 0) THEN
			Temperatures.eTempSensPT100	:=	TCond;
		ELSIF (FIND(str1:=stSensName, str2:='TAmb') <> 0) THEN
			Temperatures.eTempSensPT100	:=	TAmb;
		END_IF
		nIndSens	:=	Temperatures.eTempSensPT100;
	ELSE
		Step	:=	90;
	END_IF	
	
	fbReader.eCmd	:=	eEnumCmd_Next;	//Read next value (slope)
	fbReader(pBuffer:=ADR(sLine), cbBuffer:=SIZEOF(sLine));
	
	IF fbReader.bOk THEN
		Temperatures.stTempSensPT100[nIndSens].fParaM := STRING_TO_REAL(fbReader.getValue);
	ELSE
		Step	:=	90;
	END_IF	
	
	fbReader.eCmd	:=	eEnumCmd_Next;	//Read next value (offset)
	fbReader(pBuffer:=ADR(sLine), cbBuffer:=SIZEOF(sLine));
	
	IF fbReader.bOk THEN
		Temperatures.stTempSensPT100[nIndSens].fParaC := STRING_TO_REAL(fbReader.getValue); //account for header
	ELSE
		Step	:=	90;
	END_IF
	
	fbReader.eCmd	:=	eEnumCmd_Next;	//Read next value (maximum value)
	fbReader(pBuffer:=ADR(sLine), cbBuffer:=SIZEOF(sLine));
	
	IF fbReader.bOk THEN
		Temperatures.stTempSensPT100[nIndSens].fParaMaxVal := STRING_TO_REAL(fbReader.getValue); //account for header
	ELSE
		Step	:=	90;
	END_IF
	
	fbReader.eCmd	:=	eEnumCmd_Next;	//Read next value (minimum value)
	fbReader(pBuffer:=ADR(sLine), cbBuffer:=SIZEOF(sLine));
	
	IF fbReader.bOk THEN
		Temperatures.stTempSensPT100[nIndSens].fParaMinVal := STRING_TO_REAL(fbReader.getValue);
	ELSE
		Step	:=	90;
	END_IF
	
	//Read next line
	Step	:=	3;
	
10:	//end of csv file
	IF (hFile <> 0) THEN
		Step	:=	20; //close file
	END_IF
	
20:	//close csv file
	fbFileClose(bExecute:=FALSE);
	fbFileClose(sNetId:='', hFile:=hFile, bExecute:=TRUE, tTimeout:=T#5S);
	Step	:=	21;
	
21:	
	fbFileClose(bExecute:=FALSE);
	IF NOT fbFileClose.bBusy THEN
		step	:=	0;	//Standby mode
		bCompleted	:=	TRUE;
	END_IF
	
90:	//TODO: Error handling
	bError	:=	TRUE;
	IF (hFile <> 0) THEN
		Step	:=	20;	//close file
	END_IF

END_CASE

END_FUNCTION_BLOCK

// ---- POUs/Initialize/FB_ReadTempResTabVR11.TcPOU
FUNCTION_BLOCK FB_ReadTempResTabVR11
VAR_INPUT
	bExecute		:	BOOL	:= FALSE;
END_VAR
VAR_OUTPUT
	bCompleted		:	BOOL	:=	FALSE;
	bError			:	BOOL	:=	FALSE;
END_VAR
VAR
	fbFileOpen		:	FB_FileOpen;
	fbFileGets		:	FB_FileGets;
	fbReader		:	FB_CSVMemBufferReader;
	fbFileClose		:	FB_FileClose;
	sCSVPath		:	STRING	:=	'D:\cve-mme\WpPruefstandData\KennlinieVR11.csv';	//Path to csv file
	hFile			:	UINT;
	bEOF			:	BOOL	:=	FALSE;
	Step			:	DWORD	:=	0;
	sLine			:	STRING;	//Line read by fbFileGets
	nLine			:	UINT	:=	0;
END_VAR

CASE Step OF
	
0:	//Standby mode
	IF bExecute THEN
		bExecute	:=	FALSE; //reset to defaults
		hFile		:=	0;
		bEOF		:=	FALSE;
		bCompleted	:=	FALSE;
		bError		:=	FALSE;
		sLine		:=	'';
		nLine		:=	0;
		Step		:=	1; //start program
	END_IF

1:	//Open file
	fbFileOpen(sNetId:='', sPathName:=sCSVPath, nMode:=FOPEN_MODEREAD OR FOPEN_MODETEXT,
		ePath:=PATH_GENERIC, tTimeout:=T#5s, bExecute:=TRUE);
	Step	:=	Step + 1;

2:
	fbFileOpen(bExecute:=FALSE);
	IF NOT fbFileOpen.bBusy THEN
		IF NOT fbFileOpen.bError THEN
			//Store file handle
			hFile	:=	fbFileOpen.hFile;
			Step	:=	Step + 1;
		ELSE
			Step	:=	90;	
		END_IF
	END_IF

3:	//Read csv file
	fbFileGets(sNetId:='', hFile:=hFile, bExecute:=TRUE, tTimeout:=T#5S);
	nLine	:=	nLine + 1;
	Step	:=	Step + 1;

4:
	fbFileGets(bExecute:=FALSE);
	IF NOT fbFileGets.bBusy THEN
		IF NOT (nLine = 1) THEN //Header -> jump to next line
			IF NOT fbFileGets.bError THEN
				IF fbFileGets.bEOF THEN
					Step	:=	10; //Reached end of file
				ELSE
					sLine	:=	fbFileGets.sLine; //store line
					IF RIGHT(sLine,1) = '$L' THEN
						sLine	:=	REPLACE(sLINE, '$R$L', 2, LEN(sLine)); //restore CRLF characters
					END_IF
					Step	:=	Step + 1;
				END_IF
			ELSE
				Step	:=	90;
			END_IF
		ELSE
			Step	:=	3;
		END_IF
	END_IF
	
5:	//Parse line
	
	fbReader.eCmd	:=	eEnumCmd_First;	//Read first value (temperature)
	fbReader(pBuffer:=ADR(sLine), cbBuffer:=SIZEOF(sLine));
	
	IF fbReader.bOk THEN
		TempConvDat.VR11[nLine-1,2] := STRING_TO_REAL(fbReader.getValue);	//account for header
	ELSE
		Step	:=	90;
	END_IF	
	
	fbReader.eCmd	:=	eEnumCmd_Next;	//Read next value (resistance)
	fbReader(pBuffer:=ADR(sLine), cbBuffer:=SIZEOF(sLine));
	
	IF fbReader.bOk THEN
		TempConvDat.VR11[nLine-1,1] := STRING_TO_REAL(fbReader.getValue); //account for header
	ELSE
		Step	:=	90;
	END_IF
	
	//Read next line
	Step	:=	3;
	
10:	//end of csv file
	IF (hFile <> 0) THEN
		Step	:=	20; //close file
	END_IF
	
20:	//close csv file
	fbFileClose(bExecute:=FALSE);
	fbFileClose(sNetId:='', hFile:=hFile, bExecute:=TRUE, tTimeout:=T#5S);
	Step	:=	21;
	
21:	
	fbFileClose(bExecute:=FALSE);
	IF NOT fbFileClose.bBusy THEN
		step	:=	0;	//Standby mode
		bCompleted	:=	TRUE;
	END_IF
	
90:	//TODO: Error handling
	bError	:=	TRUE;
	IF (hFile <> 0) THEN
		Step	:=	20;	//close file
	END_IF

END_CASE

END_FUNCTION_BLOCK

// ---- POUs/Initialize/P_InitMain.TcPOU
PROGRAM P_InitMain
VAR
	bComplete	:	BOOL	:=	FALSE;
	bError		:	BOOL	:=	FALSE;
	fbInitTimes				:	FB_InitTimes;
	fbReadTempResTabVR10	:	FB_ReadTempResTabVR10;
	fbReadTempResTabVR11	:	FB_ReadTempResTabVR11;
	fbReadPressTab			:	FB_ReadPressTab;	
	fbReadPt100Tab			:	FB_ReadPT100Tab;
	fbPumpTimes				:	FB_InitPumpTimes;
	fbHeatCurve				:	FB_ReadHeatCurve;
	fbNightMode				:	FB_ReadNightMode;
END_VAR

//Initialization program
IF NOT fbInitTimes.bReady THEN
	fbInitTimes();
END_IF

IF NOT fbPumpTimes.bReady THEN	//only once
	fbPumpTimes();
END_IF

IF NOT fbNightMode.bCompleted THEN
	fbNightMode(bExecute:=TRUE);
END_IF

//set initial values for pumps -> 0.75V: no pump operation
AnaOutputs.stOutpBP.fVal	:=	0.75;
AnaOutputs.stOutpExtHP.fVal	:=	0.75;
AnaOutputs.stOutpIntHP.fVal	:=	0.75;

//Read temperature sensor data from csv-files
IF NOT fbReadTempResTabVR10.bCompleted THEN
	fbReadTempResTabVR10(bExecute:=TRUE);
END_IF
IF NOT fbReadTempResTabVR11.bCompleted THEN
	fbReadTempResTabVR11(bExecute:=TRUE);
END_IF
IF NOT fbReadPressTab.bCompleted THEN
	fbReadPressTab(bExecute:=TRUE);
END_IF
IF NOT fbReadPT100Tab.bCompleted THEN
	fbReadPT100Tab(bExecute:=TRUE);
END_IF
IF NOT fbHeatCurve.bCompleted THEN
	fbHeatCurve(bExecute:=TRUE);
END_IF

IF fbReadTempResTabVR10.bCompleted AND fbReadTempResTabVR11.bCompleted AND fbReadPressTab.bCompleted 
		AND fbReadPT100Tab.bCompleted AND fbInitTimes.bReady AND fbHeatCurve.bCompleted AND fbNightMode.bCompleted THEN
	bComplete	:=	TRUE;
END_IF

IF fbReadTempResTabVR10.bError OR fbReadTempResTabVR11.bError OR fbReadPressTab.bError 
		OR fbReadPT100Tab.bError OR fbHeatCurve.bError OR fbNightMode.bError THEN
	bError		:=	TRUE;
END_IF

END_PROGRAM

// ---- POUs/Initialize/FB_ReadTempResTabVR10.TcPOU
FUNCTION_BLOCK FB_ReadTempResTabVR10
VAR_INPUT
	bExecute		:	BOOL	:= FALSE;
END_VAR
VAR_OUTPUT
	bCompleted		:	BOOL	:=	FALSE;
	bError			:	BOOL	:=	FALSE;
END_VAR
VAR
	fbFileOpen		:	FB_FileOpen;
	fbFileGets		:	FB_FileGets;
	fbReader		:	FB_CSVMemBufferReader;
	fbFileClose		:	FB_FileClose;
	sCSVPath		:	STRING	:=	'D:\cve-mme\WpPruefstandData\KennlinieVR10.csv';	//Path to csv file
	hFile			:	UINT;
	bEOF			:	BOOL	:=	FALSE;
	Step			:	DWORD	:=	0;
	sLine			:	STRING;	//Line read by fbFileGets
	nLine			:	UINT	:=	0;
END_VAR

CASE Step OF
	
0:	//Standby mode
	IF bExecute THEN
		bExecute	:=	FALSE; //reset to defaults
		hFile		:=	0;
		bEOF		:=	FALSE;
		bCompleted	:=	FALSE;
		bError		:=	FALSE;
		sLine		:=	'';
		nLine		:=	0;
		Step		:=	1; //start program
	END_IF

1:	//Open file
	fbFileOpen(sNetId:='', sPathName:=sCSVPath, nMode:=FOPEN_MODEREAD OR FOPEN_MODETEXT,
		ePath:=PATH_GENERIC, tTimeout:=T#5s, bExecute:=TRUE);
	Step	:=	Step + 1;

2:
	fbFileOpen(bExecute:=FALSE);
	IF NOT fbFileOpen.bBusy THEN
		IF NOT fbFileOpen.bError THEN
			//Store file handle
			hFile	:=	fbFileOpen.hFile;
			Step	:=	Step + 1;
		ELSE
			Step	:=	90;	
		END_IF
	END_IF

3:	//Read csv file
	fbFileGets(sNetId:='', hFile:=hFile, bExecute:=TRUE, tTimeout:=T#5S);
	nLine	:=	nLine + 1;
	Step	:=	Step + 1;

4:
	fbFileGets(bExecute:=FALSE);
	IF NOT fbFileGets.bBusy THEN
		IF NOT (nLine = 1) THEN //Header -> jump to next line
			IF NOT fbFileGets.bError THEN
				IF fbFileGets.bEOF THEN
					Step	:=	10; //Reached end of file
				ELSE
					sLine	:=	fbFileGets.sLine; //store line
					IF RIGHT(sLine,1) = '$L' THEN
						sLine	:=	REPLACE(sLINE, '$R$L', 2, LEN(sLine)); //restore CRLF characters
					END_IF
					Step	:=	Step + 1;
				END_IF
			ELSE
				Step	:=	90;
			END_IF
		ELSE
			Step	:=	3;
		END_IF
	END_IF
	
5:	//Parse line
	
	fbReader.eCmd	:=	eEnumCmd_First;	//Read first value (temperature)
	fbReader(pBuffer:=ADR(sLine), cbBuffer:=SIZEOF(sLine));
	
	IF fbReader.bOk THEN
		TempConvDat.VR10[nLine-1,2] := STRING_TO_REAL(fbReader.getValue);	//account for header
	ELSE
		Step	:=	90;
	END_IF	
	
	fbReader.eCmd	:=	eEnumCmd_Next;	//Read next value (resistance)
	fbReader(pBuffer:=ADR(sLine), cbBuffer:=SIZEOF(sLine));
	
	IF fbReader.bOk THEN
		TempConvDat.VR10[nLine-1,1] := STRING_TO_REAL(fbReader.getValue); //account for header
	ELSE
		Step	:=	90;
	END_IF
	
	//Read next line
	Step	:=	3;
	
10:	//end of csv file
	IF (hFile <> 0) THEN
		Step	:=	20; //close file
	END_IF
	
20:	//close csv file
	fbFileClose(bExecute:=FALSE);
	fbFileClose(sNetId:='', hFile:=hFile, bExecute:=TRUE, tTimeout:=T#5S);
	Step	:=	21;
	
21:	
	fbFileClose(bExecute:=FALSE);
	IF NOT fbFileClose.bBusy THEN
		step	:=	0;	//Standby mode
		bCompleted	:=	TRUE;
	END_IF
	
90:	//TODO: Error handling
	bError	:=	TRUE;
	IF (hFile <> 0) THEN
		Step	:=	20;	//close file
	END_IF

END_CASE

END_FUNCTION_BLOCK

// ---- POUs/Read/F_LinSens.TcPOU
FUNCTION F_LinSens	:	ST_InputVar
VAR_INPUT
	stInput	:	ST_InputVar;
END_VAR
VAR
END_VAR

stInput.fVal	:=	stInput.fParaM * DINT_TO_REAL(stInput.nVarInput) + stInput.fParaC; //linear conversion

IF stInput.bSensErr THEN
	stInput.bValid	:=	FALSE;
END_IF

//check if value is valid
IF (stInput.fVal > stInput.fParaMaxVal) OR (stInput.fVal < stInput.fParaMinVal) THEN
	stInput.bValid	:=	FALSE;
END_IF

F_LinSens	:=	stInput;	//return

END_FUNCTION

// ---- POUs/Read/P_PowMeas.TcPOU
PROGRAM P_PowMeas
VAR
END_VAR

//Total effective power = sum of effective power of phases
PowMeas.fEffPow		:=	PowMeas.stPowMeas[0].fEffPow + PowMeas.stPowMeas[1].fEffPow + PowMeas.stPowMeas[2].fEffPow;
//Mean power factor
PowMeas.fMeanCosPhi	:=	(PowMeas.stPowMeas[0].fcosPhi * PowMeas.stPowMeas[1].fcosPhi * PowMeas.stPowMeas[2].fcosPhi) / 3;
//Power factor = effective power / apparent power
IF (PowMeas.fMeanCosPhi <> 0) THEN
	PowMeas.fAppPow		:=	PowMeas.fEffPow / PowMeas.fMeanCosPhi;
END_IF
//Apparent power = sqrt(effective power^2 + reaktive power^2)
PowMeas.fReaPow		:= SQRT((PowMeas.fAppPow * PowMeas.fAppPow) - (PowMeas.fEffPow * PowMeas.fEffPow));

END_PROGRAM

// ---- POUs/Read/P_ReadMain.TcPOU
PROGRAM P_ReadMain
VAR
	ePress		: 	E_PRESS;
	ePT100		:	E_TempSensPT100;
	eVR10		:	E_TempSensVR10;
	eVR11		:	E_TempSensVR11;
	ePowMeas	:	E_PowMeas;
END_VAR

//Read pressure sensors
FOR ePress := HP TO BP DO
	Pressures.stPress[ePress]	:=	F_LinSens(stInput:=Pressures.stPress[ePress]);
END_FOR

//Read PT100 sensors
FOR ePT100 := TExpVEv TO TAmb DO
	Temperatures.stTempSensPT100[ePT100]	:=	F_LinSens(stInput:=Temperatures.stTempSensPT100[ePT100]);
END_FOR

//Read VR10 sensors
FOR eVR10 := SP TO RF1 DO
	Temperatures.stTempSensVR10[eVR10]	:=	F_NTCSens(stInput:=Temperatures.stTempSensVR10[eVR10], pIntTab:=ADR(TempConvDat.VR10));
END_FOR

//Read VR11 sensors
FOR eVR11 := T1 TO T8 DO
	Temperatures.stTempSensVR11[eVR11]	:=	F_NTCSens(stInput:=Temperatures.stTempSensVR11[eVR11], pIntTab:=ADR(TempConvDat.VR11));
END_FOR

//Read power measurement phase values
FOR ePowMeas := L1 TO L3 DO
	PowMeas.stPowMeas[ePowMeas]	:=	F_PowMeasPhase(stInput:=PowMeas.stPowMeas[ePowMeas]);
END_FOR
//Calculate accumulated power values
P_PowMeas();

END_PROGRAM

// ---- POUs/SystemCheck/F_CheckCompCycPress.TcPOU
FUNCTION F_CheckCompCycPress : BOOL
VAR_INPUT
END_VAR
VAR
	eHP			:	E_Press	:=	HP;
	eLP			:	E_Press	:=	LP;
	bCompCycF	:	BOOL	:=	FALSE;
END_VAR

bCompCycF	:=	FALSE;

//check compression cycle pressures
IF Pressures.stPress[eHP].fVal > SysCheckParams.fHPMax THEN
	bCompCycF				:=	TRUE;
	StateMachine.bFault		:=	TRUE;
	StateMachine.nFault		:=	45;
	StateMachine.sFaultMess	:=	'Compression cycle: Pressure too high';
END_IF

IF Pressures.stPress[eLP].fVal < SysCheckParams.fLPMin THEN
	bCompCycF				:=	TRUE;
	StateMachine.bFault		:=	TRUE;
	StateMachine.nFault		:=	46;
	StateMachine.sFaultMess	:=	'Compression cycle: Pressure too low';
END_IF

IF (Pressures.stPress[eLP].fVal > (SysCheckParams.fLPMin + 0.5)) AND (Pressures.stPress[eHP].fVal < (SysCheckParams.fHPMax - 0.5)) THEN
	bCompCycF	:=	FALSE;
END_IF

END_FUNCTION

// ---- POUs/SystemCheck/F_CheckCompOutTemp.TcPOU
FUNCTION F_CheckCompOutTemp : BOOL
VAR_INPUT
END_VAR
VAR
	eT1				:	E_TempSensVR11	:=	T1;
	bCompOutTempF	:	BOOL			:=	FALSE;
END_VAR

bCompOutTempF	:=	FALSE;

//check compressor outlet temperature
IF Temperatures.stTempSensVR11[eT1].fVal > SysCheckParams.fTempCompOutMax THEN
	bCompOutTempF	:=	TRUE;
	StateMachine.bFault		:=	TRUE;
	StateMachine.nFault		:=	21;
	StateMachine.sFaultMess	:=	'Compressor outlet temperature too high';
END_IF

IF Temperatures.stTempSensVR11[eT1].fVal < (SysCheckParams.fTempCompOutMax - 2) THEN
	bCompOutTempF	:=	FALSE;
END_IF

//assign output
F_CheckCompOutTemp	:=	bCompOutTempF;

END_FUNCTION

// ---- POUs/SystemCheck/F_CheckHeatCirPress.TcPOU
FUNCTION F_CheckHeatCirPress : BOOL
VAR_INPUT
END_VAR
VAR
	eHCP		:	E_Press	:=	HCP;
	bHCPF		:	BOOL	:=	FALSE;
END_VAR

//check heating circuit pressure
IF Pressures.stPress[eHCP].fVal < SysCheckParams.fHCPMinOff THEN
	bHCPF					:=	TRUE;
	StateMachine.bFault		:=	TRUE;
	StateMachine.nFault		:=	44;
	StateMachine.sFaultMess	:=	'Heating circuit pressure too low';
END_IF

IF Pressures.stPress[eHCP].fVal > SysCheckParams.fHCPMinOn THEN
	bHCPF			:=	FALSE;
	(*
	Do not reset StateMachine fault here, in case there are other system faults!
	*)
END_IF

//assign output
F_CheckHeatCirPress	:=	bHCPF;

END_FUNCTION

// ---- POUs/SystemCheck/P_SysCheckMain.TcPOU
PROGRAM P_SysCheckMain
VAR
END_VAR

//check real-time communication with terminals (working counter wc)
SysCheck.bTermErrRT	:=	F_CheckTerm();

//check sensors
SysCheck.bSensErr	:=	F_CheckSens();

//check operating conditions
SysCheck.bAmbTemp	:=	F_CheckAmbTemp();
SysCheck.bBP			:=	F_CheckBrinePressure();
SysCheck.bHCP		:=	F_CheckHeatCirPress();

//check compression cycle pressures
SysCheck.bCompCyc	:=	F_CheckCompCycPress();

//check phase sequence
SysCheck.bPhaseSeqCh:=	F_CheckPhaseSeq();

//check heating circuit temperatures
SysCheck.bHeatTemp	:=	F_CheckHeatCirTemp();

//check compressor outlet temperature
SysCheck.bCompOut	:=	F_CheckCompOutTemp();

END_PROGRAM

// ---- POUs/Write/P_WriteMain.TcPOU
PROGRAM P_WriteMain
VAR
	fbRampBP			:	FB_RampPump;
	fbRampIntHeatC		:	FB_RampPump;
	fbRampExtHeatC		:	FB_RampPump;
	fValBPNew			:	REAL;
	fValIntHeatCPumpNew	:	REAL;
	fValExtHeatCPumpNew	:	REAL;
	tTimeToMax			:	Time	:=	T#10s;
END_VAR

//write digital outputs
DigOutputs.bOutpComp		:=	StateMachine.bCompRun;
DigOutputs.bOutpAH			:=	StateMachine.bAuxHeatOp;
DigOutputs.bSHDHWSwitchValv	:=	StateMachine.bSwitchVal;

//prepare values for analog outputs
IF StateMachine.bBrinePump THEN	//operate brine pump
	fValBPNew	:=	F_PumpConvPercVolt(StateMachine.nBrinePump);
ELSE	//stop brine pump
	fValBPNew	:=	0.75;		//0.5-1V: pump stops
END_IF
IF (AnaOutputs.stOutpBP.fVal <> fValBPNew) THEN	//old value <> new value -> ramp
	IF NOT fbRampBP.bActiveRamp THEN	//initialize
		fbRampBP.fStartVal	:=	AnaOutputs.stOutpBP.fVal;
		fbRampBP.fEndVal	:=	fValBPNew;
		//allow 10s to get to maximum speed
		fbRampBP.tDuration	:=	REAL_TO_TIME((ABS(AnaOutputs.stOutpBP.fVal - fValBPNew)/10) * TIME_TO_REAL(tTimeToMax));
		fbRampBP();	//execute function block
		AnaOutputs.stOutpBP.fVal	:=	fbRampBP.fCurVal;	//pass current value to output
	ELSE
		fbRampBP();	//execute function block
		AnaOutputs.stOutpBP.fVal	:=	fbRampBP.fCurVal;	//pass current value to output
	END_IF
ELSE
	AnaOutputs.stOutpBP.fVal	:=	fValBPNew;
END_IF

IF StateMachine.bIntHeatCPump THEN	//operate internal heating circuit pump
	fValIntHeatCPumpNew	:=	F_PumpConvPercVolt(StateMachine.nIntHeatCPump);
ELSE	//stop internal heating circuit pump
	fValIntHeatCPumpNew	:=	0.75;		//0.5-1V: pump stops
END_IF
IF (AnaOutputs.stOutpIntHP.fVal <> fValIntHeatCPumpNew) THEN	//old value <> new value -> ramp
	IF NOT fbRampIntHeatC.bActiveRamp THEN	//initialize
		fbRampIntHeatC.fStartVal	:=	AnaOutputs.stOutpIntHP.fVal;
		fbRampIntHeatC.fEndVal		:=	fValIntHeatCPumpNew;
		//allow 10s to get to maximum speed
		fbRampIntHeatC.tDuration	:=	REAL_TO_TIME((ABS(AnaOutputs.stOutpIntHP.fVal - fValIntHeatCPumpNew)/10) * TIME_TO_REAL(tTimeToMax));
		fbRampIntHeatC();	//execute function block
		AnaOutputs.stOutpIntHP.fVal	:=	fbRampIntHeatC.fCurVal;	//pass current value to output
	ELSE
		fbRampIntHeatC();	//execute function block
		AnaOutputs.stOutpIntHP.fVal	:=	fbRampIntHeatC.fCurVal;	//pass current value to output
	END_IF
ELSE
	AnaOutputs.stOutpIntHP.fVal	:=	fValIntHeatCPumpNew;
END_IF

IF StateMachine.bExtHeatCPump THEN	//operate external heating circuit pump
	fValExtHeatCPumpNew	:=	F_PumpConvPercVolt(StateMachine.nExtHeatCPump);
ELSE	//stop External heating circuit pump
	fValExtHeatCPumpNew	:=	0.75;		//0.5-1V: pump stops
END_IF
IF (AnaOutputs.stOutpExtHP.fVal <> fValExtHeatCPumpNew) THEN	//old value <> new value -> ramp
	IF NOT fbRampExtHeatC.bActiveRamp THEN	//initialize
		fbRampExtHeatC.fStartVal	:=	AnaOutputs.stOutpExtHP.fVal;
		fbRampExtHeatC.fEndVal		:=	fValExtHeatCPumpNew;
		//allow 10s to get to maximum speed
		fbRampExtHeatC.tDuration	:=	REAL_TO_TIME((ABS(AnaOutputs.stOutpExtHP.fVal - fValExtHeatCPumpNew)/10) * TIME_TO_REAL(tTimeToMax));
		fbRampExtHeatC();	//execute function block
		AnaOutputs.stOutpExtHP.fVal	:=	fbRampExtHeatC.fCurVal;	//pass current value to output
	ELSE
		fbRampExtHeatC();	//execute function block
		AnaOutputs.stOutpExtHP.fVal	:=	fbRampExtHeatC.fCurVal;	//pass current value to output
	END_IF
ELSE
	AnaOutputs.stOutpExtHP.fVal	:=	fValExtHeatCPumpNew;
END_IF

AnaOutputs.stOutpMixValv.fVal	:=	StateMachine.fMixVal;

//convert voltages to int signals and write to terminal
AnaOutputs.stOutpBP			:=	F_ConvLinAnaOutp(stOutput:=AnaOutputs.stOutpBP);
AnaOutputs.stOutpIntHP		:=	F_ConvLinAnaOutp(stOutput:=AnaOutputs.stOutpIntHP);
AnaOutputs.stOutpExtHP		:=	F_ConvLinAnaOutp(stOutput:=AnaOutputs.stOutpExtHP);
AnaOutputs.stOutpMixValv	:=	F_ConvLinAnaOutp(stOutput:=AnaOutputs.stOutpMixValv);

END_PROGRAM
